(* IEC 61131-3 sources: RL_MAR/experiments/comparison/autoplc/results/gpt-4o_20260511_211137/med_27, 1 file *)

(* ---- med_27_1.st ---- *)
FUNCTION_BLOCK FlowerArrangingMachine
VAR_INPUT
    FlowerTypeSensor : INT; (* Input for detecting flower type *)
    FlowerColorSensor : INT; (* Input for detecting flower color *)
END_VAR
VAR_OUTPUT
    ArrangingMechanism : INT; (* Output for controlling arranging mechanism *)
    ConveyorBelt : BOOL; (* Output for controlling conveyor belt *)
END_VAR

VAR
    isRedType1 : BOOL;
    isBlueType1 : BOOL;
    isRedType2 : BOOL;
    isBlueType2 : BOOL;
END_VAR

(* Control logic to determine the state of the arranging mechanism and conveyor belt *)
IF (FlowerTypeSensor = 1) AND (FlowerColorSensor = 1) THEN
    ArrangingMechanism := 1;
ELSIF (FlowerTypeSensor = 1) AND (FlowerColorSensor = 2) THEN
    ArrangingMechanism := 2;
ELSIF (FlowerTypeSensor = 2) AND (FlowerColorSensor = 1) THEN
    ArrangingMechanism := 3;
ELSIF (FlowerTypeSensor = 2) AND (FlowerColorSensor = 2) THEN
    ArrangingMechanism := 4;
ELSE
    ArrangingMechanism := 0;
END_IF;

(* Control logic for the conveyor belt based on the arranging mechanism state *)
IF ArrangingMechanism <> 0 THEN
    ConveyorBelt := TRUE;
ELSE
    ConveyorBelt := FALSE;
END_IF;

END_FUNCTION_BLOCK
